FUNCTION_BLOCK ChangeDetect (* Basic Function Block Type *)
  (* Standard: 61499-2 *)
  (* Version 0.0, 5/28/2016, Andrei, nxtControl GmbH, Template *)
  PACKAGE Main;
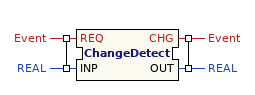
  EVENT_INPUT
    REQ WITH INP; (* Normal Execution Request *)
  END_EVENT
  EVENT_OUTPUT
    CHG WITH OUT; (* Execution Confirmation *)
  END_EVENT
  VAR_INPUT
    INP : REAL; (* Input event qualifier *)
  END_VAR
  VAR_OUTPUT
    OUT : REAL; (* Output event qualifier *)
  END_VAR
  VAR
    PREV : REAL;
  END_VAR
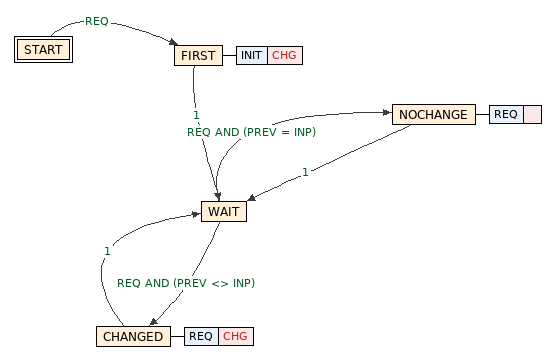
  EC_STATES
    START; (* Initial State *)
    NOCHANGE : REQ; (* Initialization *)
    CHANGED : REQ -> CHG; (* Normal execution *)
    WAIT;
    FIRST : INIT -> CHG;
  END_STATES
  EC_TRANSITIONS
    WAIT TO NOCHANGE := REQ AND (PREV = INP);
    NOCHANGE TO WAIT := 1;
    WAIT TO CHANGED := REQ AND (PREV <> INP);
    CHANGED TO WAIT := 1;
    FIRST TO WAIT := 1;
    START TO FIRST := REQ;
  END_TRANSITIONS
  ALGORITHM INIT IN ST: (* Initialization algorithm *)
PREV:=INP;
OUT:=INP;
  END_ALGORITHM
  ALGORITHM REQ IN ST: (* Normally executed algorithm *)
PREV := INP;
OUT := INP;
  END_ALGORITHM
END_FUNCTION_BLOCK
